FUNCTION_BLOCK FB_WaterController IMPLEMENTS I_WaterController

VAR
	bInletValve : BOOL;
	bOutletValve : BOOL;
	
	tBaseTime : TIME := T#5S;
	tFillingTime : TIME ;
	tDrainingTime : TIME ;
	
	fbWaterTimer : TON;
END_VAR

METHOD GetDuration : TIME
VAR_INPUT
	stWash : REFERENCE TO ST_Wash;
END_VAR

tFillingTime := tBaseTime * stWash.nWaterLevel;
tDrainingTime := tBaseTime * stWash.nWaterLevel;
GetDuration := tFillingTime + tDrainingTime;
END_METHOD

{warning 'add method implementation '}
METHOD StartDrain : BOOL

StartDrain := bOutletValve := TRUE;
fbWaterTimer( IN := bOutletValve, PT := tFillingTime);
IF fbWaterTimer.Q THEN
	bOutletValve := FALSE;
	StartDrain := FALSE;
	fbWaterTimer( IN := bOutletValve);
END_IF
END_METHOD

{warning 'add method implementation '}
METHOD StartFill : BOOL
bInletValve := TRUE;
fbWaterTimer( IN := bInletValve, PT := tFillingTime);
IF fbWaterTimer.Q THEN
	bInletValve := FALSE;
	StartFill := TRUE;
	fbWaterTimer( IN := bInletValve);
END_IF
END_METHOD

METHOD Stop : BOOL
VAR_INPUT
END_VAR
bInletValve := bOutletValve := FALSE;
END_METHOD

END_FUNCTION_BLOCK

(* stored: Version 1.1.0.1, ProductVersion 3.1.4024.16
   POU FB_WaterController: Id {7607c710-6c9a-4822-8ef3-44a38a1af84a}, SpecialFunc None
   Method GetDuration: Id {d6c6978b-fca7-424e-b214-ba7165bb22b2}
   Method StartDrain: Id {e16c08f7-9931-405a-b27b-99e175bb7de5}
   Method StartFill: Id {486a3f2d-fad5-4077-a4a6-f327b9894499}
   Method Stop: Id {5fc106ba-0ed7-49a2-81c6-6d53439a16ca} *)
